// TIA Portal project "iodevice" (V15)

(* hardware
DEVICE "S71500/ET200MP station_1"  S7-1500 station
   slot 0: "Rail_0"  Rack  6ES7 590-1***0-0AA0
   slot 1: "PLC_1"  CPU 1511-1 PN  6ES7 511-1AK00-0AB0  V1.8
      slot 3: "CPU display_1"  6ES7591-1AA00-0AA0
   slot 2: "AI/AQ 4xU/I/RTD/TC / 2xU/I ST_1"  AI/AQ 4xU/I/RTD/TC / 2xU/I ST  6ES7 534-7QE00-0AB0  V1.0
*)

// ===== PLC "PLC_1"  CPU 1511-1 PN =====

VAR_GLOBAL   // PLC tag table "Default tag table"
   "trigger" AT %Q0.0 : Bool;
   "output" AT %Q0.1 : Bool;
   "inturpt" AT %Q0.2 : Bool;
   "genIN" AT %Q0.3 : Bool;
   "genOUT" AT %Q0.4 : Bool;
   "in1" AT %M0.0 : Bool;
   "out1" AT %M0.1 : Bool;
   "out2" AT %M0.2 : Bool;
   "out3" AT %M0.3 : Bool;
   "out3count" AT %MW2 : Int;
   "out1count" AT %MW4 : Int;
END_VAR

DATA_BLOCK "lad2_DB"   // DB1
{ S7_Optimized_Access := 'TRUE' }
VERSION : 0.1
// stored: InstanceOfName lad2
"lad2"
BEGIN
END_DATA_BLOCK

// folder: System blocks/Program resources

DATA_BLOCK "IEC_Counter_0_DB"   // DB2
{ S7_Optimized_Access := 'TRUE' }
AUTHOR : Simatic
FAMILY : IEC
NAME : CNTR
VERSION : 1.0
// stored: InstanceOfName IEC_COUNTER
"IEC_COUNTER"
BEGIN
END_DATA_BLOCK

DATA_BLOCK "IEC_Counter_0_DB_1"   // DB3
{ S7_Optimized_Access := 'TRUE' }
AUTHOR : Simatic
FAMILY : IEC
NAME : CNTR
VERSION : 1.0
// stored: InstanceOfName IEC_COUNTER
"IEC_COUNTER"
BEGIN
END_DATA_BLOCK

// folder: (top level)

FUNCTION_BLOCK "lad2"   // FB1, LAD
{ S7_Optimized_Access := 'TRUE' }
VERSION : 0.1
   VAR
      ONS : Bool;
   END_VAR
   VAR_TEMP   // added for the SCL form of the ladder/FBD networks
      _w1 : Bool;
   END_VAR
BEGIN

REGION Network 1
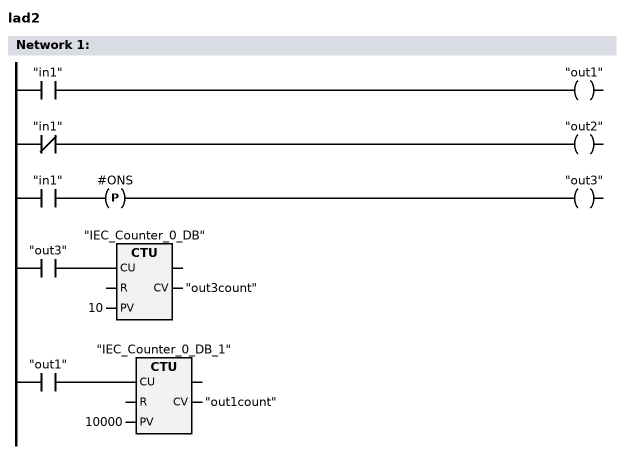
   "out1" := "in1";
   "out2" := NOT "in1";
   #_w1 := "in1" AND NOT #ONS;   // rising edge
   #ONS := "in1";
   "out3" := #_w1;
   "IEC_Counter_0_DB".CTU(CU := "out3", PV := 10, CV => "out3count");
   "IEC_Counter_0_DB_1".CTU(CU := "out1", PV := 10000, CV => "out1count");
END_REGION
END_FUNCTION_BLOCK

ORGANIZATION_BLOCK "Main"   // OB1, LAD, ProgramCycle
TITLE = "Main Program Sweep (Cycle)"
{ S7_Optimized_Access := 'TRUE' }
VERSION : 0.1
   VAR_INPUT
      Initial_Call : Bool;   // Initial call of this OB
      Remanence : Bool;   // =True, if remanent data are available
   END_VAR
BEGIN

REGION Network 1
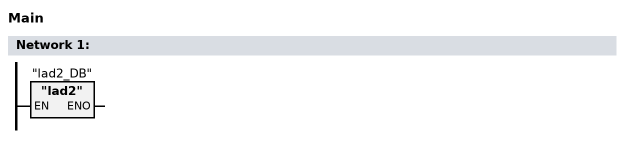
   RUNG wire#powerrail
      "lad2_DB"()
   END_RUNG
   // the same network as SCL:
   "lad2_DB"();   // "lad2"
END_REGION
END_ORGANIZATION_BLOCK